Staubli VAL3: OMAC_Unhold.pgx

program OMAC_Unhold()
  local joint l_jHere
begin
  //OMAC进程:UnHolding
  _nOmacStat=7
  logMsg("上位机手动操作：恢复")
  resetMotion()
  call trackErr_init()
  enablePower()
  l_jHere=herej()
  l_jHere.j3=jHome.j3
  movej(l_jHere,tGripper,mSlow)
  movej(jHome,tGripper,mSlow)
  _bSentToHome=true
  waitEndMove()
  if taskStatus("cellManager")>=0
    taskKill("cellManager")
  endIf
  wait(taskStatus("cellManager")<0)
  taskCreate "cellManager",100,cellManager()
  wait(taskStatus("cellManager")==1)

  delay(0)
end
